// Mitsubishi GX Developer project: パレット移載装置   PLC: Q02

PROGRAM SENSOR
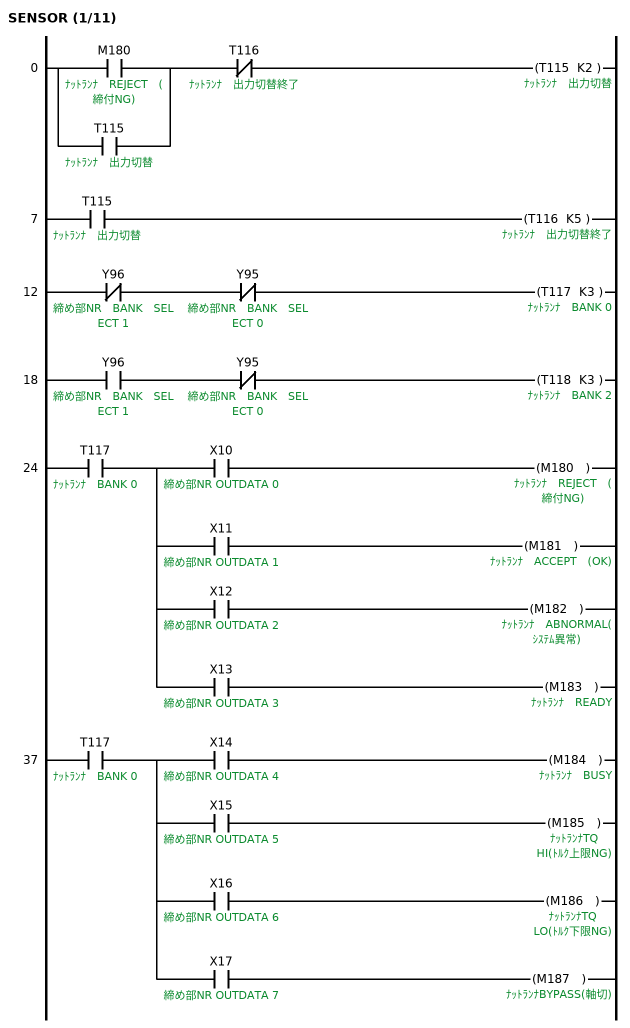
0     LD      M180  ; ﾅｯﾄﾗﾝﾅ　REJECT　(締付NG)
      OR      T115  ; ﾅｯﾄﾗﾝﾅ　出力切替
      ANI     T116  ; ﾅｯﾄﾗﾝﾅ　出力切替終了
      OUT     T115 K2  ; ﾅｯﾄﾗﾝﾅ　出力切替
7     LD      T115  ; ﾅｯﾄﾗﾝﾅ　出力切替
      OUT     T116 K5  ; ﾅｯﾄﾗﾝﾅ　出力切替終了
12    LDI     Y96  ; 締め部NR　BANK　SELECT 1
      ANI     Y95  ; 締め部NR　BANK　SELECT 0
      OUT     T117 K3  ; ﾅｯﾄﾗﾝﾅ　BANK 0
18    LD      Y96  ; 締め部NR　BANK　SELECT 1
      ANI     Y95  ; 締め部NR　BANK　SELECT 0
      OUT     T118 K3  ; ﾅｯﾄﾗﾝﾅ　BANK 2
24    LD      T117  ; ﾅｯﾄﾗﾝﾅ　BANK 0
      MPS
      AND     X10  ; 締め部NR OUTDATA 0
      OUT     M180  ; ﾅｯﾄﾗﾝﾅ　REJECT　(締付NG)
      MRD
      AND     X11  ; 締め部NR OUTDATA 1
      OUT     M181  ; ﾅｯﾄﾗﾝﾅ　ACCEPT　(OK)
      MRD
      AND     X12  ; 締め部NR OUTDATA 2
      OUT     M182  ; ﾅｯﾄﾗﾝﾅ　ABNORMAL(ｼｽﾃﾑ異常)
      MPP
      AND     X13  ; 締め部NR OUTDATA 3
      OUT     M183  ; ﾅｯﾄﾗﾝﾅ　READY
37    LD      T117  ; ﾅｯﾄﾗﾝﾅ　BANK 0
      MPS
      AND     X14  ; 締め部NR OUTDATA 4
      OUT     M184  ; ﾅｯﾄﾗﾝﾅ　BUSY
      MRD
      AND     X15  ; 締め部NR OUTDATA 5
      OUT     M185  ; ﾅｯﾄﾗﾝﾅTQ HI(ﾄﾙｸ上限NG)
      MRD
      AND     X16  ; 締め部NR OUTDATA 6
      OUT     M186  ; ﾅｯﾄﾗﾝﾅTQ LO(ﾄﾙｸ下限NG)
      MPP
      AND     X17  ; 締め部NR OUTDATA 7
      OUT     M187  ; ﾅｯﾄﾗﾝﾅBYPASS(軸切)
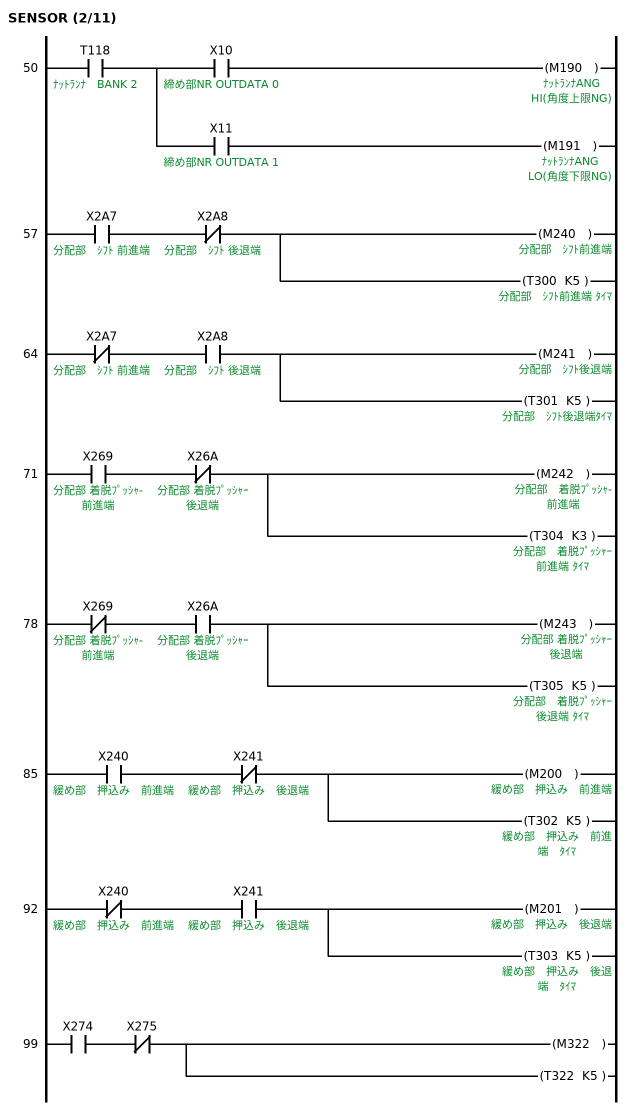
50    LD      T118  ; ﾅｯﾄﾗﾝﾅ　BANK 2
      MPS
      AND     X10  ; 締め部NR OUTDATA 0
      OUT     M190  ; ﾅｯﾄﾗﾝﾅANG HI(角度上限NG)
      MPP
      AND     X11  ; 締め部NR OUTDATA 1
      OUT     M191  ; ﾅｯﾄﾗﾝﾅANG LO(角度下限NG)
57    LD      X2A7  ; 分配部　ｼﾌﾄ 前進端
      ANI     X2A8  ; 分配部　ｼﾌﾄ 後退端
      OUT     M240  ; 分配部　ｼﾌﾄ前進端
      OUT     T300 K5  ; 分配部　ｼﾌﾄ前進端 ﾀｲﾏ
64    LDI     X2A7  ; 分配部　ｼﾌﾄ 前進端
      AND     X2A8  ; 分配部　ｼﾌﾄ 後退端
      OUT     M241  ; 分配部　ｼﾌﾄ後退端
      OUT     T301 K5  ; 分配部　ｼﾌﾄ後退端ﾀｲﾏ
71    LD      X269  ; 分配部 着脱ﾌﾟｯｼｬ- 前進端
      ANI     X26A  ; 分配部 着脱ﾌﾟｯｼｬｰ 後退端
      OUT     M242  ; 分配部　着脱ﾌﾟｯｼｬ- 前進端
      OUT     T304 K3  ; 分配部　着脱ﾌﾟｯｼｬｰ 前進端 ﾀｲﾏ
78    LDI     X269  ; 分配部 着脱ﾌﾟｯｼｬ- 前進端
      AND     X26A  ; 分配部 着脱ﾌﾟｯｼｬｰ 後退端
      OUT     M243  ; 分配部 着脱ﾌﾟｯｼｬｰ 後退端
      OUT     T305 K5  ; 分配部　着脱ﾌﾟｯｼｬｰ 後退端 ﾀｲﾏ
85    LD      X240  ; 緩め部　押込み　前進端
      ANI     X241  ; 緩め部　押込み　後退端
      OUT     M200  ; 緩め部　押込み　前進端
      OUT     T302 K5  ; 緩め部　押込み　前進端　ﾀｲﾏ
92    LDI     X240  ; 緩め部　押込み　前進端
      AND     X241  ; 緩め部　押込み　後退端
      OUT     M201  ; 緩め部　押込み　後退端
      OUT     T303 K5  ; 緩め部　押込み　後退端　ﾀｲﾏ
99    LD      X274
      ANI     X275
      OUT     M322
      OUT     T322 K5
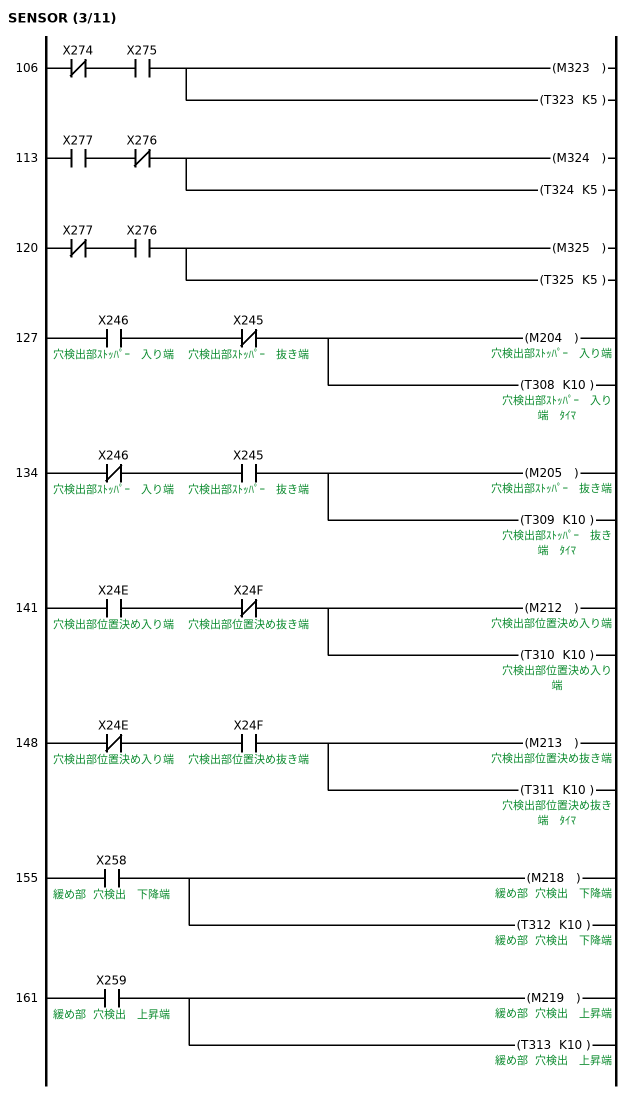
106   LDI     X274
      AND     X275
      OUT     M323
      OUT     T323 K5
113   LD      X277
      ANI     X276
      OUT     M324
      OUT     T324 K5
120   LDI     X277
      AND     X276
      OUT     M325
      OUT     T325 K5
127   LD      X246  ; 穴検出部ｽﾄｯﾊﾟｰ　入り端
      ANI     X245  ; 穴検出部ｽﾄｯﾊﾟｰ　抜き端
      OUT     M204  ; 穴検出部ｽﾄｯﾊﾟｰ　入り端
      OUT     T308 K10  ; 穴検出部ｽﾄｯﾊﾟｰ　入り端　ﾀｲﾏ
134   LDI     X246  ; 穴検出部ｽﾄｯﾊﾟｰ　入り端
      AND     X245  ; 穴検出部ｽﾄｯﾊﾟｰ　抜き端
      OUT     M205  ; 穴検出部ｽﾄｯﾊﾟｰ　抜き端
      OUT     T309 K10  ; 穴検出部ｽﾄｯﾊﾟｰ　抜き端　ﾀｲﾏ
141   LD      X24E  ; 穴検出部位置決め入り端
      ANI     X24F  ; 穴検出部位置決め抜き端
      OUT     M212  ; 穴検出部位置決め入り端
      OUT     T310 K10  ; 穴検出部位置決め入り端
148   LDI     X24E  ; 穴検出部位置決め入り端
      AND     X24F  ; 穴検出部位置決め抜き端
      OUT     M213  ; 穴検出部位置決め抜き端
      OUT     T311 K10  ; 穴検出部位置決め抜き端　ﾀｲﾏ
155   LD      X258  ; 緩め部  穴検出　下降端
      OUT     M218  ; 緩め部  穴検出　下降端
      OUT     T312 K10  ; 緩め部  穴検出　下降端
161   LD      X259  ; 緩め部  穴検出　上昇端
      OUT     M219  ; 緩め部  穴検出　上昇端
      OUT     T313 K10  ; 緩め部  穴検出　上昇端
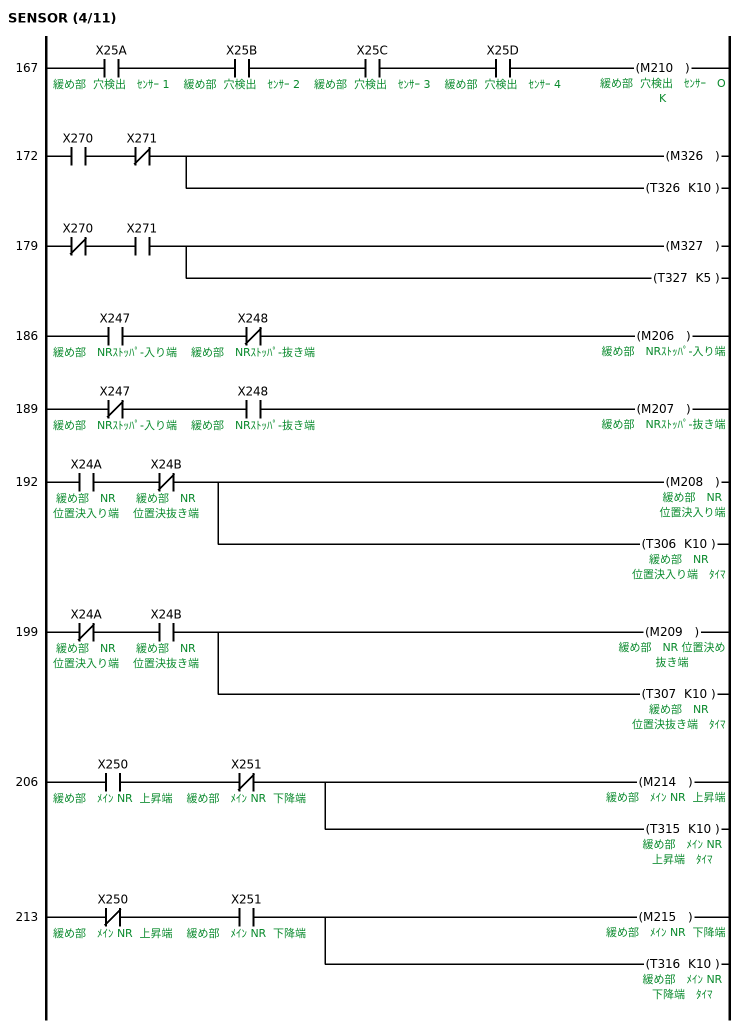
167   LD      X25A  ; 緩め部  穴検出　ｾﾝｻｰ 1
      AND     X25B  ; 緩め部  穴検出　ｾﾝｻｰ 2
      AND     X25C  ; 緩め部  穴検出　ｾﾝｻｰ 3
      AND     X25D  ; 緩め部  穴検出　ｾﾝｻｰ 4
      OUT     M210  ; 緩め部  穴検出　ｾﾝｻｰ　OK
172   LD      X270
      ANI     X271
      OUT     M326
      OUT     T326 K10
179   LDI     X270
      AND     X271
      OUT     M327
      OUT     T327 K5
186   LD      X247  ; 緩め部　NRｽﾄｯﾊﾟ-入り端
      ANI     X248  ; 緩め部　NRｽﾄｯﾊﾟ-抜き端
      OUT     M206  ; 緩め部　NRｽﾄｯﾊﾟ-入り端
189   LDI     X247  ; 緩め部　NRｽﾄｯﾊﾟ-入り端
      AND     X248  ; 緩め部　NRｽﾄｯﾊﾟ-抜き端
      OUT     M207  ; 緩め部　NRｽﾄｯﾊﾟ-抜き端
192   LD      X24A  ; 緩め部　NR 位置決入り端
      ANI     X24B  ; 緩め部　NR 位置決抜き端
      OUT     M208  ; 緩め部　NR 位置決入り端
      OUT     T306 K10  ; 緩め部　NR 位置決入り端　ﾀｲﾏ
199   LDI     X24A  ; 緩め部　NR 位置決入り端
      AND     X24B  ; 緩め部　NR 位置決抜き端
      OUT     M209  ; 緩め部　NR 位置決め 抜き端
      OUT     T307 K10  ; 緩め部　NR 位置決抜き端　ﾀｲﾏ
206   LD      X250  ; 緩め部　ﾒｲﾝ NR  上昇端
      ANI     X251  ; 緩め部　ﾒｲﾝ NR  下降端
      OUT     M214  ; 緩め部　ﾒｲﾝ NR  上昇端
      OUT     T315 K10  ; 緩め部　ﾒｲﾝ NR  上昇端　ﾀｲﾏ
213   LDI     X250  ; 緩め部　ﾒｲﾝ NR  上昇端
      AND     X251  ; 緩め部　ﾒｲﾝ NR  下降端
      OUT     M215  ; 緩め部　ﾒｲﾝ NR  下降端
      OUT     T316 K10  ; 緩め部　ﾒｲﾝ NR  下降端　ﾀｲﾏ
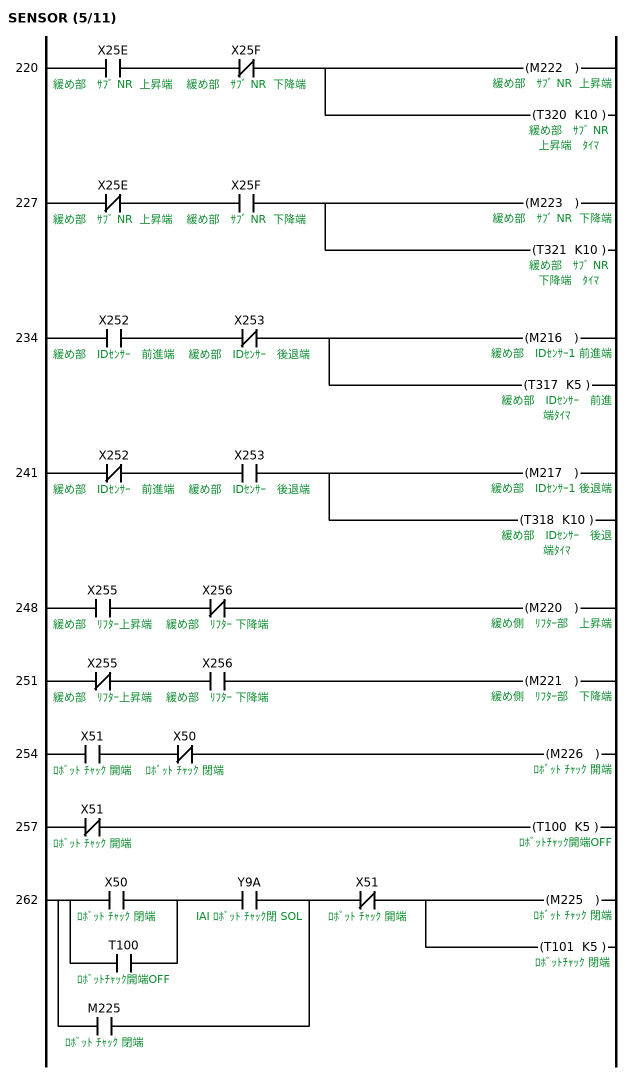
220   LD      X25E  ; 緩め部　ｻﾌﾞ NR  上昇端
      ANI     X25F  ; 緩め部　ｻﾌﾞ NR  下降端
      OUT     M222  ; 緩め部　ｻﾌﾞ NR  上昇端
      OUT     T320 K10  ; 緩め部　ｻﾌﾞ NR  上昇端　ﾀｲﾏ
227   LDI     X25E  ; 緩め部　ｻﾌﾞ NR  上昇端
      AND     X25F  ; 緩め部　ｻﾌﾞ NR  下降端
      OUT     M223  ; 緩め部　ｻﾌﾞ NR  下降端
      OUT     T321 K10  ; 緩め部　ｻﾌﾞ NR  下降端　ﾀｲﾏ
234   LD      X252  ; 緩め部　IDｾﾝｻｰ　前進端
      ANI     X253  ; 緩め部　IDｾﾝｻｰ　後退端
      OUT     M216  ; 緩め部　IDｾﾝｻｰ1 前進端
      OUT     T317 K5  ; 緩め部　IDｾﾝｻｰ　前進端ﾀｲﾏ
241   LDI     X252  ; 緩め部　IDｾﾝｻｰ　前進端
      AND     X253  ; 緩め部　IDｾﾝｻｰ　後退端
      OUT     M217  ; 緩め部　IDｾﾝｻｰ1 後退端
      OUT     T318 K10  ; 緩め部　IDｾﾝｻｰ　後退端ﾀｲﾏ
248   LD      X255  ; 緩め部　ﾘﾌﾀｰ上昇端
      ANI     X256  ; 緩め部　ﾘﾌﾀｰ 下降端
      OUT     M220  ; 緩め側　ﾘﾌﾀｰ部　上昇端
251   LDI     X255  ; 緩め部　ﾘﾌﾀｰ上昇端
      AND     X256  ; 緩め部　ﾘﾌﾀｰ 下降端
      OUT     M221  ; 緩め側　ﾘﾌﾀｰ部　下降端
254   LD      X51  ; ﾛﾎﾞｯﾄ ﾁｬｯｸ 開端
      ANI     X50  ; ﾛﾎﾞｯﾄ ﾁｬｯｸ 閉端
      OUT     M226  ; ﾛﾎﾞｯﾄ ﾁｬｯｸ 開端
257   LDI     X51  ; ﾛﾎﾞｯﾄ ﾁｬｯｸ 開端
      OUT     T100 K5  ; ﾛﾎﾞｯﾄﾁｬｯｸ開端OFF
262   LD      X50  ; ﾛﾎﾞｯﾄ ﾁｬｯｸ 閉端
      OR      T100  ; ﾛﾎﾞｯﾄﾁｬｯｸ開端OFF
      AND     Y9A  ; IAI ﾛﾎﾞｯﾄ ﾁｬｯｸ閉 SOL
      OR      M225  ; ﾛﾎﾞｯﾄ ﾁｬｯｸ 閉端
      ANI     X51  ; ﾛﾎﾞｯﾄ ﾁｬｯｸ 開端
      OUT     M225  ; ﾛﾎﾞｯﾄ ﾁｬｯｸ 閉端
      OUT     T101 K5  ; ﾛﾎﾞｯﾄﾁｬｯｸ 閉端
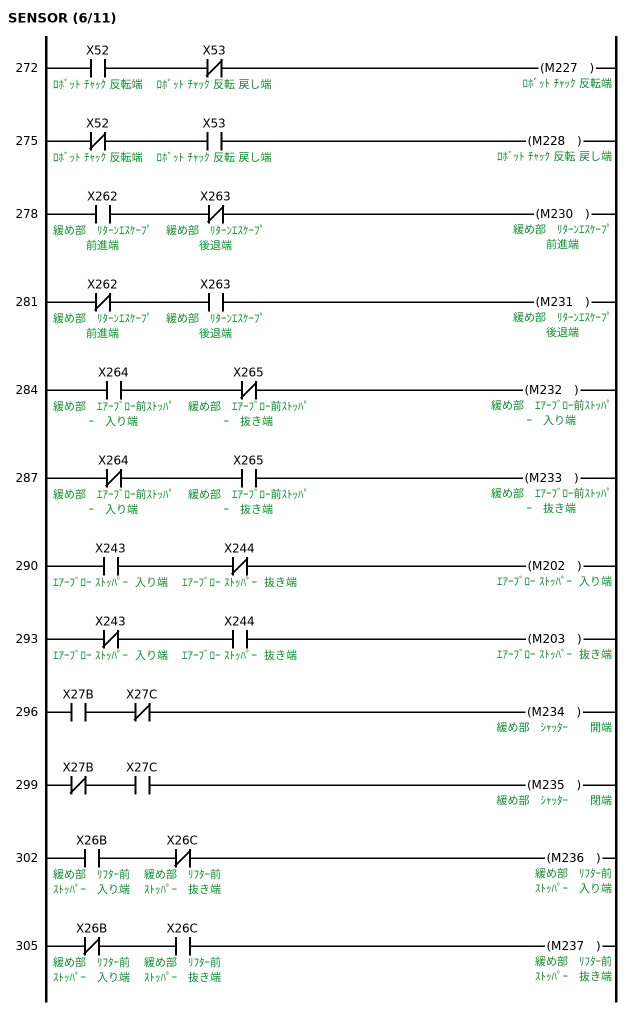
272   LD      X52  ; ﾛﾎﾞｯﾄ ﾁｬｯｸ 反転端
      ANI     X53  ; ﾛﾎﾞｯﾄ ﾁｬｯｸ 反転 戻し端
      OUT     M227  ; ﾛﾎﾞｯﾄ ﾁｬｯｸ 反転端
275   LDI     X52  ; ﾛﾎﾞｯﾄ ﾁｬｯｸ 反転端
      AND     X53  ; ﾛﾎﾞｯﾄ ﾁｬｯｸ 反転 戻し端
      OUT     M228  ; ﾛﾎﾞｯﾄ ﾁｬｯｸ 反転 戻し端
278   LD      X262  ; 緩め部　ﾘﾀｰﾝｴｽｹｰﾌﾟ 前進端
      ANI     X263  ; 緩め部　ﾘﾀｰﾝｴｽｹｰﾌﾟ 後退端
      OUT     M230  ; 緩め部　ﾘﾀｰﾝｴｽｹｰﾌﾟ 前進端
281   LDI     X262  ; 緩め部　ﾘﾀｰﾝｴｽｹｰﾌﾟ 前進端
      AND     X263  ; 緩め部　ﾘﾀｰﾝｴｽｹｰﾌﾟ 後退端
      OUT     M231  ; 緩め部　ﾘﾀｰﾝｴｽｹｰﾌﾟ 後退端
284   LD      X264  ; 緩め部　ｴｱｰﾌﾞﾛｰ前ｽﾄｯﾊﾟｰ　入り端
      ANI     X265  ; 緩め部　ｴｱｰﾌﾞﾛｰ前ｽﾄｯﾊﾟｰ　抜き端
      OUT     M232  ; 緩め部　ｴｱｰﾌﾞﾛｰ前ｽﾄｯﾊﾟｰ　入り端
287   LDI     X264  ; 緩め部　ｴｱｰﾌﾞﾛｰ前ｽﾄｯﾊﾟｰ　入り端
      AND     X265  ; 緩め部　ｴｱｰﾌﾞﾛｰ前ｽﾄｯﾊﾟｰ　抜き端
      OUT     M233  ; 緩め部　ｴｱｰﾌﾞﾛｰ前ｽﾄｯﾊﾟｰ　抜き端
290   LD      X243  ; ｴｱｰﾌﾞﾛｰ ｽﾄｯﾊﾟｰ  入り端
      ANI     X244  ; ｴｱｰﾌﾞﾛｰ ｽﾄｯﾊﾟｰ  抜き端
      OUT     M202  ; ｴｱｰﾌﾞﾛｰ ｽﾄｯﾊﾟｰ  入り端
293   LDI     X243  ; ｴｱｰﾌﾞﾛｰ ｽﾄｯﾊﾟｰ  入り端
      AND     X244  ; ｴｱｰﾌﾞﾛｰ ｽﾄｯﾊﾟｰ  抜き端
      OUT     M203  ; ｴｱｰﾌﾞﾛｰ ｽﾄｯﾊﾟｰ  抜き端
296   LD      X27B
      ANI     X27C
      OUT     M234  ; 緩め部　ｼｬｯﾀｰ　　開端
299   LDI     X27B
      AND     X27C
      OUT     M235  ; 緩め部　ｼｬｯﾀｰ　　閉端
302   LD      X26B  ; 緩め部　ﾘﾌﾀｰ前  ｽﾄｯﾊﾟｰ　入り端
      ANI     X26C  ; 緩め部　ﾘﾌﾀｰ前  ｽﾄｯﾊﾟｰ　抜き端
      OUT     M236  ; 緩め部　ﾘﾌﾀｰ前  ｽﾄｯﾊﾟｰ　入り端
305   LDI     X26B  ; 緩め部　ﾘﾌﾀｰ前  ｽﾄｯﾊﾟｰ　入り端
      AND     X26C  ; 緩め部　ﾘﾌﾀｰ前  ｽﾄｯﾊﾟｰ　抜き端
      OUT     M237  ; 緩め部　ﾘﾌﾀｰ前  ｽﾄｯﾊﾟｰ　抜き端
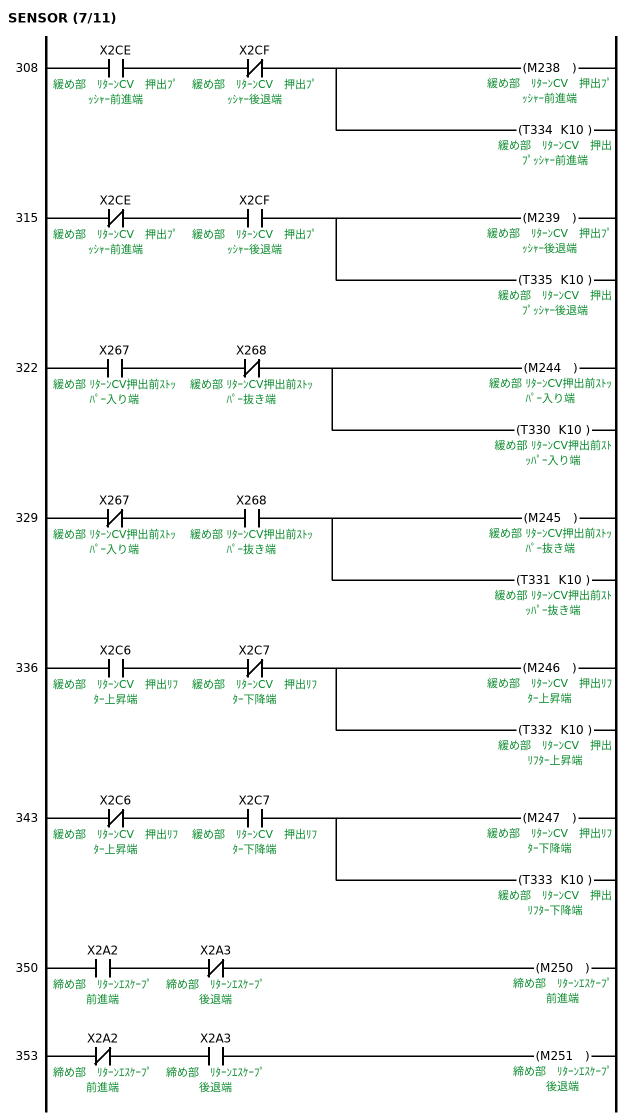
308   LD      X2CE  ; 緩め部　ﾘﾀｰﾝCV　押出ﾌﾟｯｼｬｰ前進端
      ANI     X2CF  ; 緩め部　ﾘﾀｰﾝCV　押出ﾌﾟｯｼｬｰ後退端
      OUT     M238  ; 緩め部　ﾘﾀｰﾝCV　押出ﾌﾟｯｼｬｰ前進端
      OUT     T334 K10  ; 緩め部　ﾘﾀｰﾝCV　押出ﾌﾟｯｼｬｰ前進端
315   LDI     X2CE  ; 緩め部　ﾘﾀｰﾝCV　押出ﾌﾟｯｼｬｰ前進端
      AND     X2CF  ; 緩め部　ﾘﾀｰﾝCV　押出ﾌﾟｯｼｬｰ後退端
      OUT     M239  ; 緩め部　ﾘﾀｰﾝCV　押出ﾌﾟｯｼｬｰ後退端
      OUT     T335 K10  ; 緩め部　ﾘﾀｰﾝCV　押出ﾌﾟｯｼｬｰ後退端
322   LD      X267  ; 緩め部 ﾘﾀｰﾝCV押出前ｽﾄｯﾊﾟｰ入り端
      ANI     X268  ; 緩め部 ﾘﾀｰﾝCV押出前ｽﾄｯﾊﾟｰ抜き端
      OUT     M244  ; 緩め部 ﾘﾀｰﾝCV押出前ｽﾄｯﾊﾟｰ入り端
      OUT     T330 K10  ; 緩め部 ﾘﾀｰﾝCV押出前ｽﾄｯﾊﾟｰ入り端
329   LDI     X267  ; 緩め部 ﾘﾀｰﾝCV押出前ｽﾄｯﾊﾟｰ入り端
      AND     X268  ; 緩め部 ﾘﾀｰﾝCV押出前ｽﾄｯﾊﾟｰ抜き端
      OUT     M245  ; 緩め部 ﾘﾀｰﾝCV押出前ｽﾄｯﾊﾟｰ抜き端
      OUT     T331 K10  ; 緩め部 ﾘﾀｰﾝCV押出前ｽﾄｯﾊﾟｰ抜き端
336   LD      X2C6  ; 緩め部　ﾘﾀｰﾝCV　押出ﾘﾌﾀｰ上昇端
      ANI     X2C7  ; 緩め部　ﾘﾀｰﾝCV　押出ﾘﾌﾀｰ下降端
      OUT     M246  ; 緩め部　ﾘﾀｰﾝCV　押出ﾘﾌﾀｰ上昇端
      OUT     T332 K10  ; 緩め部　ﾘﾀｰﾝCV　押出ﾘﾌﾀｰ上昇端
343   LDI     X2C6  ; 緩め部　ﾘﾀｰﾝCV　押出ﾘﾌﾀｰ上昇端
      AND     X2C7  ; 緩め部　ﾘﾀｰﾝCV　押出ﾘﾌﾀｰ下降端
      OUT     M247  ; 緩め部　ﾘﾀｰﾝCV　押出ﾘﾌﾀｰ下降端
      OUT     T333 K10  ; 緩め部　ﾘﾀｰﾝCV　押出ﾘﾌﾀｰ下降端
350   LD      X2A2  ; 締め部　ﾘﾀｰﾝｴｽｹｰﾌﾟ 前進端
      ANI     X2A3  ; 締め部　ﾘﾀｰﾝｴｽｹｰﾌﾟ 後退端
      OUT     M250  ; 締め部　ﾘﾀｰﾝｴｽｹｰﾌﾟ 前進端
353   LDI     X2A2  ; 締め部　ﾘﾀｰﾝｴｽｹｰﾌﾟ 前進端
      AND     X2A3  ; 締め部　ﾘﾀｰﾝｴｽｹｰﾌﾟ 後退端
      OUT     M251  ; 締め部　ﾘﾀｰﾝｴｽｹｰﾌﾟ 後退端
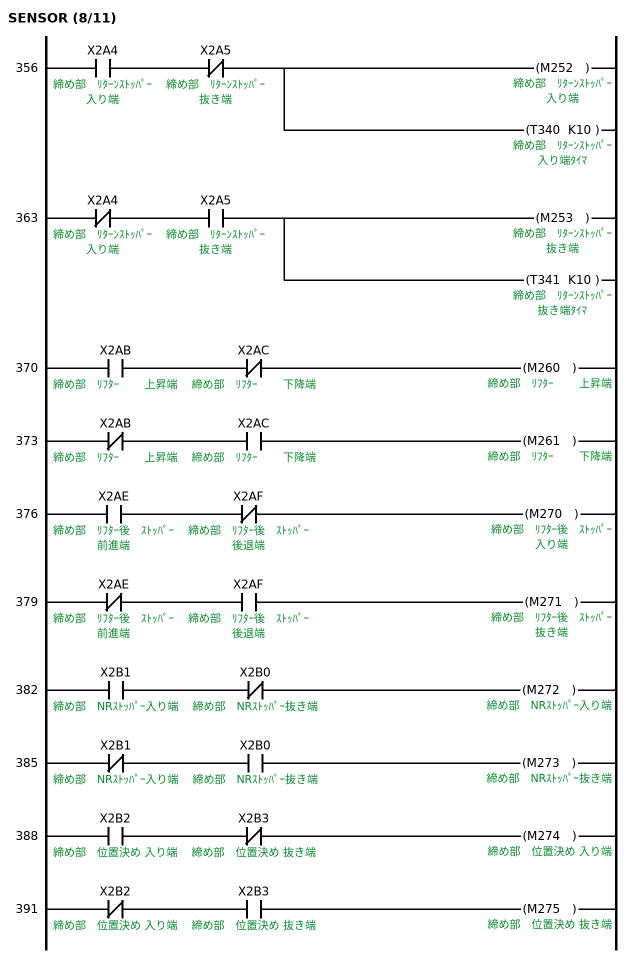
356   LD      X2A4  ; 締め部　ﾘﾀｰﾝｽﾄｯﾊﾟｰ 入り端
      ANI     X2A5  ; 締め部　ﾘﾀｰﾝｽﾄｯﾊﾟｰ 抜き端
      OUT     M252  ; 締め部　ﾘﾀｰﾝｽﾄｯﾊﾟｰ 入り端
      OUT     T340 K10  ; 締め部　ﾘﾀｰﾝｽﾄｯﾊﾟｰ 入り端ﾀｲﾏ
363   LDI     X2A4  ; 締め部　ﾘﾀｰﾝｽﾄｯﾊﾟｰ 入り端
      AND     X2A5  ; 締め部　ﾘﾀｰﾝｽﾄｯﾊﾟｰ 抜き端
      OUT     M253  ; 締め部　ﾘﾀｰﾝｽﾄｯﾊﾟｰ 抜き端
      OUT     T341 K10  ; 締め部　ﾘﾀｰﾝｽﾄｯﾊﾟｰ 抜き端ﾀｲﾏ
370   LD      X2AB  ; 締め部　ﾘﾌﾀｰ 　　上昇端
      ANI     X2AC  ; 締め部　ﾘﾌﾀｰ 　　下降端
      OUT     M260  ; 締め部　ﾘﾌﾀｰ 　　上昇端
373   LDI     X2AB  ; 締め部　ﾘﾌﾀｰ 　　上昇端
      AND     X2AC  ; 締め部　ﾘﾌﾀｰ 　　下降端
      OUT     M261  ; 締め部　ﾘﾌﾀｰ 　　下降端
376   LD      X2AE  ; 締め部　ﾘﾌﾀｰ後　ｽﾄｯﾊﾟｰ　前進端
      ANI     X2AF  ; 締め部　ﾘﾌﾀｰ後　ｽﾄｯﾊﾟｰ　後退端
      OUT     M270  ; 締め部　ﾘﾌﾀｰ後　ｽﾄｯﾊﾟｰ　入り端
379   LDI     X2AE  ; 締め部　ﾘﾌﾀｰ後　ｽﾄｯﾊﾟｰ　前進端
      AND     X2AF  ; 締め部　ﾘﾌﾀｰ後　ｽﾄｯﾊﾟｰ　後退端
      OUT     M271  ; 締め部　ﾘﾌﾀｰ後　ｽﾄｯﾊﾟｰ　抜き端
382   LD      X2B1  ; 締め部　NRｽﾄｯﾊﾟｰ入り端
      ANI     X2B0  ; 締め部　NRｽﾄｯﾊﾟｰ抜き端
      OUT     M272  ; 締め部　NRｽﾄｯﾊﾟｰ入り端
385   LDI     X2B1  ; 締め部　NRｽﾄｯﾊﾟｰ入り端
      AND     X2B0  ; 締め部　NRｽﾄｯﾊﾟｰ抜き端
      OUT     M273  ; 締め部　NRｽﾄｯﾊﾟｰ抜き端
388   LD      X2B2  ; 締め部　位置決め 入り端
      ANI     X2B3  ; 締め部　位置決め 抜き端
      OUT     M274  ; 締め部　位置決め 入り端
391   LDI     X2B2  ; 締め部　位置決め 入り端
      AND     X2B3  ; 締め部　位置決め 抜き端
      OUT     M275  ; 締め部　位置決め 抜き端
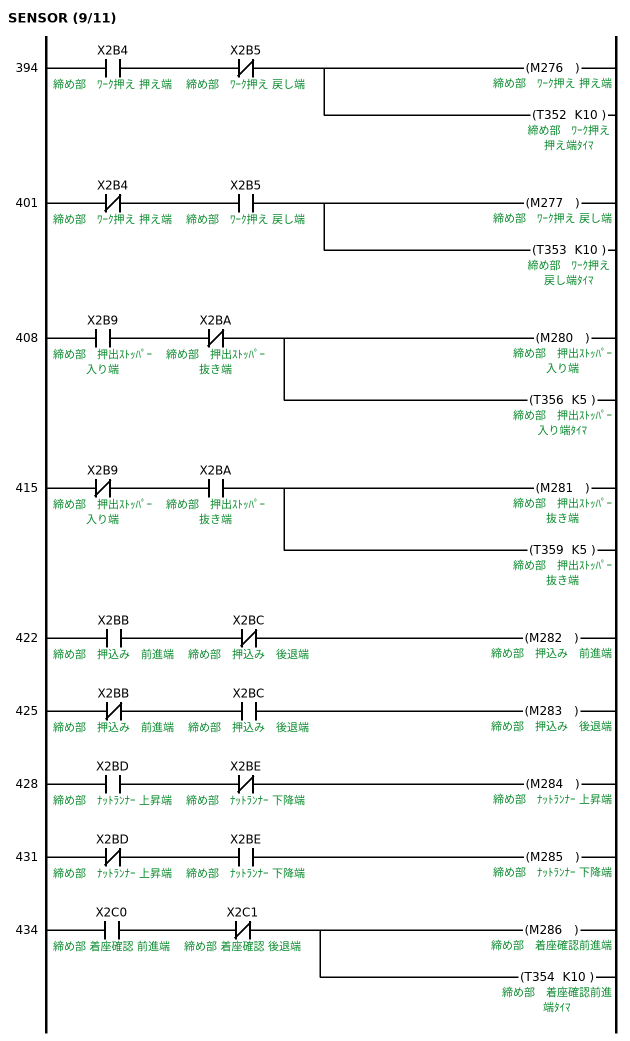
394   LD      X2B4  ; 締め部　ﾜｰｸ押え 押え端
      ANI     X2B5  ; 締め部　ﾜｰｸ押え 戻し端
      OUT     M276  ; 締め部　ﾜｰｸ押え 押え端
      OUT     T352 K10  ; 締め部　ﾜｰｸ押え 押え端ﾀｲﾏ
401   LDI     X2B4  ; 締め部　ﾜｰｸ押え 押え端
      AND     X2B5  ; 締め部　ﾜｰｸ押え 戻し端
      OUT     M277  ; 締め部　ﾜｰｸ押え 戻し端
      OUT     T353 K10  ; 締め部　ﾜｰｸ押え 戻し端ﾀｲﾏ
408   LD      X2B9  ; 締め部　押出ｽﾄｯﾊﾟｰ 入り端
      ANI     X2BA  ; 締め部　押出ｽﾄｯﾊﾟｰ 抜き端
      OUT     M280  ; 締め部　押出ｽﾄｯﾊﾟｰ 入り端
      OUT     T356 K5  ; 締め部　押出ｽﾄｯﾊﾟｰ 入り端ﾀｲﾏ
415   LDI     X2B9  ; 締め部　押出ｽﾄｯﾊﾟｰ 入り端
      AND     X2BA  ; 締め部　押出ｽﾄｯﾊﾟｰ 抜き端
      OUT     M281  ; 締め部　押出ｽﾄｯﾊﾟｰ 抜き端
      OUT     T359 K5  ; 締め部　押出ｽﾄｯﾊﾟｰ 抜き端
422   LD      X2BB  ; 締め部　押込み　前進端
      ANI     X2BC  ; 締め部　押込み　後退端
      OUT     M282  ; 締め部　押込み　前進端
425   LDI     X2BB  ; 締め部　押込み　前進端
      AND     X2BC  ; 締め部　押込み　後退端
      OUT     M283  ; 締め部　押込み　後退端
428   LD      X2BD  ; 締め部　ﾅｯﾄﾗﾝﾅｰ 上昇端
      ANI     X2BE  ; 締め部　ﾅｯﾄﾗﾝﾅｰ 下降端
      OUT     M284  ; 締め部　ﾅｯﾄﾗﾝﾅｰ 上昇端
431   LDI     X2BD  ; 締め部　ﾅｯﾄﾗﾝﾅｰ 上昇端
      AND     X2BE  ; 締め部　ﾅｯﾄﾗﾝﾅｰ 下降端
      OUT     M285  ; 締め部　ﾅｯﾄﾗﾝﾅｰ 下降端
434   LD      X2C0  ; 締め部 着座確認 前進端
      ANI     X2C1  ; 締め部 着座確認 後退端
      OUT     M286  ; 締め部　着座確認前進端
      OUT     T354 K10  ; 締め部　着座確認前進端ﾀｲﾏ
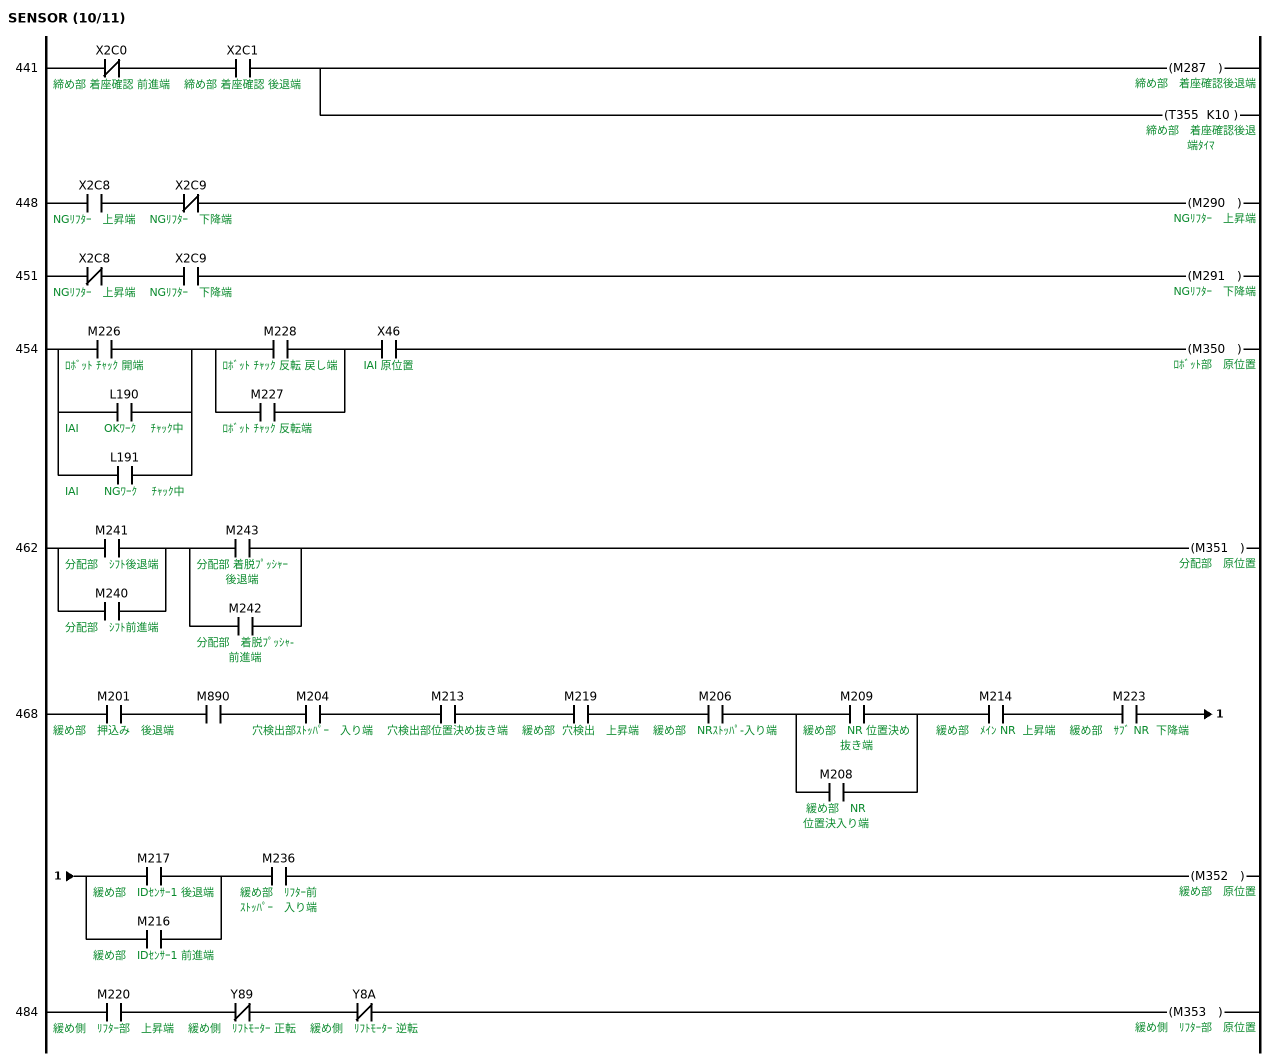
441   LDI     X2C0  ; 締め部 着座確認 前進端
      AND     X2C1  ; 締め部 着座確認 後退端
      OUT     M287  ; 締め部　着座確認後退端
      OUT     T355 K10  ; 締め部　着座確認後退端ﾀｲﾏ
448   LD      X2C8  ; NGﾘﾌﾀｰ　上昇端
      ANI     X2C9  ; NGﾘﾌﾀｰ　下降端
      OUT     M290  ; NGﾘﾌﾀｰ　上昇端
451   LDI     X2C8  ; NGﾘﾌﾀｰ　上昇端
      AND     X2C9  ; NGﾘﾌﾀｰ　下降端
      OUT     M291  ; NGﾘﾌﾀｰ　下降端
454   LD      M226  ; ﾛﾎﾞｯﾄ ﾁｬｯｸ 開端
      OR      L190  ; IAI　　 OKﾜｰｸ　 ﾁｬｯｸ中
      OR      L191  ; IAI　　 NGﾜｰｸ　 ﾁｬｯｸ中
      LD      M228  ; ﾛﾎﾞｯﾄ ﾁｬｯｸ 反転 戻し端
      OR      M227  ; ﾛﾎﾞｯﾄ ﾁｬｯｸ 反転端
      ANB
      AND     X46  ; IAI 原位置
      OUT     M350  ; ﾛﾎﾞｯﾄ部　原位置
462   LD      M241  ; 分配部　ｼﾌﾄ後退端
      OR      M240  ; 分配部　ｼﾌﾄ前進端
      LD      M243  ; 分配部 着脱ﾌﾟｯｼｬｰ 後退端
      OR      M242  ; 分配部　着脱ﾌﾟｯｼｬ- 前進端
      ANB
      OUT     M351  ; 分配部　原位置
468   LD      M201  ; 緩め部　押込み　後退端
      AND     M890
      AND     M204  ; 穴検出部ｽﾄｯﾊﾟｰ　入り端
      AND     M213  ; 穴検出部位置決め抜き端
      AND     M219  ; 緩め部  穴検出　上昇端
      AND     M206  ; 緩め部　NRｽﾄｯﾊﾟ-入り端
      LD      M209  ; 緩め部　NR 位置決め 抜き端
      OR      M208  ; 緩め部　NR 位置決入り端
      ANB
      AND     M214  ; 緩め部　ﾒｲﾝ NR  上昇端
      AND     M223  ; 緩め部　ｻﾌﾞ NR  下降端
      LD      M217  ; 緩め部　IDｾﾝｻｰ1 後退端
      OR      M216  ; 緩め部　IDｾﾝｻｰ1 前進端
      ANB
      AND     M236  ; 緩め部　ﾘﾌﾀｰ前  ｽﾄｯﾊﾟｰ　入り端
      OUT     M352  ; 緩め部　原位置
484   LD      M220  ; 緩め側　ﾘﾌﾀｰ部　上昇端
      ANI     Y89  ; 緩め側　ﾘﾌﾄﾓｰﾀｰ 正転
      ANI     Y8A  ; 緩め側　ﾘﾌﾄﾓｰﾀｰ 逆転
      OUT     M353  ; 緩め側　ﾘﾌﾀｰ部　原位置
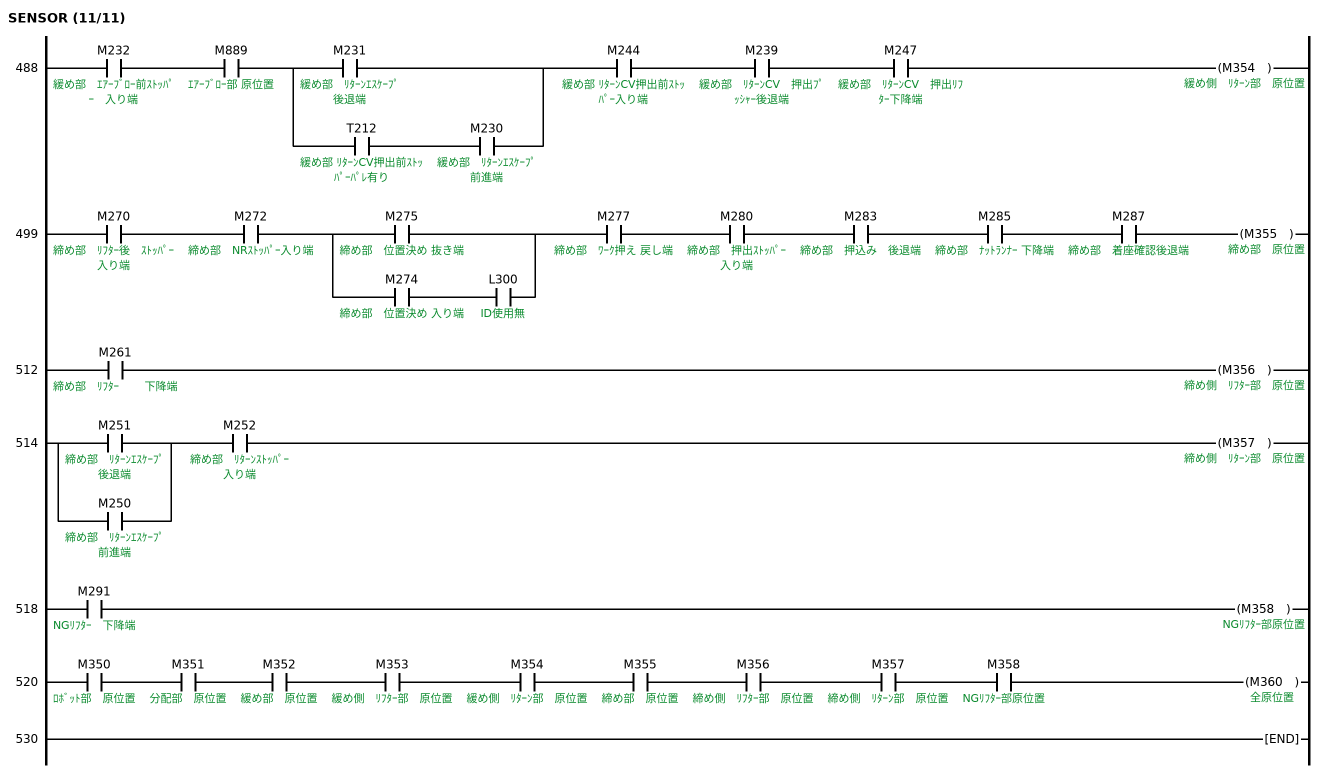
488   LD      M232  ; 緩め部　ｴｱｰﾌﾞﾛｰ前ｽﾄｯﾊﾟｰ　入り端
      AND     M889  ; ｴｱｰﾌﾞﾛｰ部 原位置
      LD      M231  ; 緩め部　ﾘﾀｰﾝｴｽｹｰﾌﾟ 後退端
      LD      T212  ; 緩め部 ﾘﾀｰﾝCV押出前ｽﾄｯﾊﾟｰﾊﾟﾚ有り
      AND     M230  ; 緩め部　ﾘﾀｰﾝｴｽｹｰﾌﾟ 前進端
      ORB
      ANB
      AND     M244  ; 緩め部 ﾘﾀｰﾝCV押出前ｽﾄｯﾊﾟｰ入り端
      AND     M239  ; 緩め部　ﾘﾀｰﾝCV　押出ﾌﾟｯｼｬｰ後退端
      AND     M247  ; 緩め部　ﾘﾀｰﾝCV　押出ﾘﾌﾀｰ下降端
      OUT     M354  ; 緩め側　ﾘﾀｰﾝ部　原位置
499   LD      M270  ; 締め部　ﾘﾌﾀｰ後　ｽﾄｯﾊﾟｰ　入り端
      AND     M272  ; 締め部　NRｽﾄｯﾊﾟｰ入り端
      LD      M275  ; 締め部　位置決め 抜き端
      LD      M274  ; 締め部　位置決め 入り端
      AND     L300  ; ID使用無
      ORB
      ANB
      AND     M277  ; 締め部　ﾜｰｸ押え 戻し端
      AND     M280  ; 締め部　押出ｽﾄｯﾊﾟｰ 入り端
      AND     M283  ; 締め部　押込み　後退端
      AND     M285  ; 締め部　ﾅｯﾄﾗﾝﾅｰ 下降端
      AND     M287  ; 締め部　着座確認後退端
      OUT     M355  ; 締め部　原位置
512   LD      M261  ; 締め部　ﾘﾌﾀｰ 　　下降端
      OUT     M356  ; 締め側　ﾘﾌﾀｰ部　原位置
514   LD      M251  ; 締め部　ﾘﾀｰﾝｴｽｹｰﾌﾟ 後退端
      OR      M250  ; 締め部　ﾘﾀｰﾝｴｽｹｰﾌﾟ 前進端
      AND     M252  ; 締め部　ﾘﾀｰﾝｽﾄｯﾊﾟｰ 入り端
      OUT     M357  ; 締め側　ﾘﾀｰﾝ部　原位置
518   LD      M291  ; NGﾘﾌﾀｰ　下降端
      OUT     M358  ; NGﾘﾌﾀｰ部原位置
520   LD      M350  ; ﾛﾎﾞｯﾄ部　原位置
      AND     M351  ; 分配部　原位置
      AND     M352  ; 緩め部　原位置
      AND     M353  ; 緩め側　ﾘﾌﾀｰ部　原位置
      AND     M354  ; 緩め側　ﾘﾀｰﾝ部　原位置
      AND     M355  ; 締め部　原位置
      AND     M356  ; 締め側　ﾘﾌﾀｰ部　原位置
      AND     M357  ; 締め側　ﾘﾀｰﾝ部　原位置
      AND     M358  ; NGﾘﾌﾀｰ部原位置
      OUT     M360  ; 全原位置
530   END
END_PROGRAM
